{attribute 'GeneratedUsingTerminal: EL5001-0000-1016'}
{attribute addProperty BoxType "EL5001-0000-1016"}
{attribute addProperty Id "EtcSlaveTerminalBaseChannel_1AT %I*Channel_DD2C734A5WcStateAT %I*WcState_9091E0EB2InfoDataAT %I*InfoData_32EB74EA10"}
{attribute addProperty CRC "3863478710"}
{attribute addProperty Size "17"}
TYPE EL5001_E64801B6 EXTENDS EtcSlaveTerminalBase :
STRUCT
	{attribute addProperty Name "Channel_1"}
	Channel_1 : Channel_DD2C734A;
	{attribute addProperty Name "WcState"}
	WcState : WcState_9091E0EB;
	{attribute addProperty Name "InfoData"}
	InfoData : InfoData_32EB74EA;
END_STRUCT
END_TYPE

(* stored: Version 1.2.0.0, ProductVersion 3.1.4024.9
   DUT EL5001_E64801B6: Id {5e158a1b-5d53-48a8-8381-73532a96742d} *)
